TYPE ST_AXIS_POS_STATUS :
STRUCT
END_STRUCT
END_TYPE

(* stored: Version 1.1.0.1, ProductVersion 3.1.4024.11
   DUT ST_AXIS_POS_STATUS: Id {e213880b-49c0-4093-9197-17ab77e77cdb} *)
